{attribute 'to_string'}
TYPE E_XPU_STATE :
(
  XTS_NULL,
  XTS_INVALID,
  XTS_INIT                      := 10,    // initialize XPU
  XTS_STATION_INFO_READ         := 20,    // get Station information from Xpu
  XTS_IDLE                      := 30
)UINT;
END_TYPE

(* stored: Version 1.1.0.1
   DUT E_XPU_STATE: Id {508f78da-6fbc-4eea-8e88-a763956d4ea1} *)
